FUNCTION F_NotEqual : BOOL
VAR_INPUT
    In1   : LREAL;
    In2   : LREAL;
    Delta : LREAL;
END_VAR
VAR
    Difference : LREAL;
END_VAR

Difference := ABS(In1 - In2);
F_NotEqual := Difference > Delta;

END_FUNCTION

(* stored: Version 1.1.0.1, ProductVersion 3.1.4024.12
   POU F_NotEqual: Id {6570352b-b3aa-47b3-b487-1de3203ea68e}, SpecialFunc None *)
